(* PLC project SafeLOGIC-1, BrAutomation SafeDESIGNER  4.3.3.7 *)
(* stored: companyURL http://www.br-automation.com, creationDateTime Fri Jan 11 12:47:24 2019 *)

PROGRAM NOTHALTKette

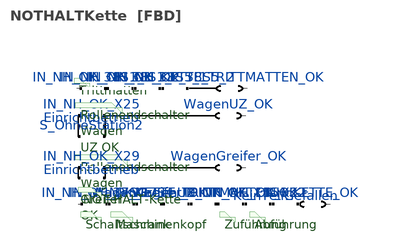
(* FBD diagram, written out as Structured Text *)
(* Trittmatten *)
NH_KETTE_TRITTMATTEN_OK := IN_NH_OK_38S1_1 AND IN_NH_OK_38S1_2 AND IN_NH_OK_38S5_1 AND IN_NH_OK_38S5_2;
(* Rollenendschalter Wagen UZ OK *)
WagenUZ_OK := IN_NH_OK_X25 OR Einrichtbetrieb OR S_OhneStation2;
(* Rollenendschalter Wagen Greifer OK *)
WagenGreifer_OK := IN_NH_OK_X29 OR Einrichtbetrieb;
(* NOT-HALT-Kette *)
NH_KETTE_OK := IN_NH_OK_37S1 AND IN_NH_OK_37S4 AND WagenGreifer_OK AND WagenUZ_OK AND NH_KETTE_TRITTMATTEN_OK AND IN_NH_OK_X15 AND IN_NH_OK_X22 AND KeinTeilGefallen;
(* Schaltschrank *)
(* Maschinenkopf *)
(* Zuführung *)
(* Abführung *)
END_PROGRAM
